(* PLC project  *)

CONFIGURATION Empty_Module_7
END_CONFIGURATION
